PROGRAM MAIN
VAR
	AIN1 AT %I*: REAL;
	OUT AT %Q*: REAL;
	Start: BOOL;
	Stop: BOOL;
	Enable AT %Q*: BOOL;
	Home: REAL;
	Measure: REAL;
	DispSet: REAL;
		
END_VAR
VAR // added by the converter: edge detectors and wires of the graphical bodies
    _w1 : BOOL;
END_VAR

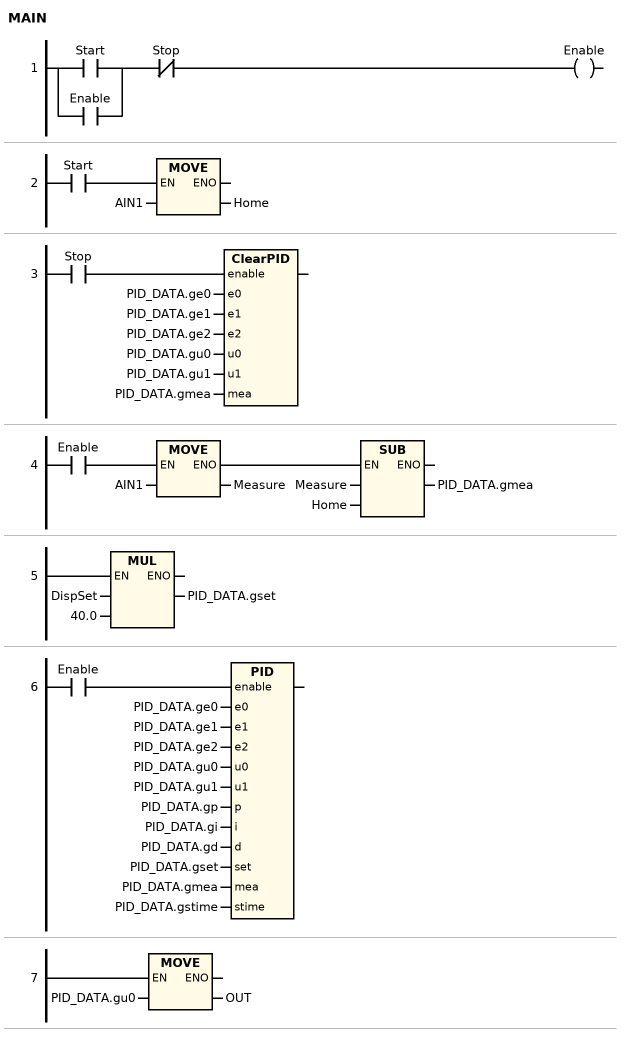
// NETWORK 1
Enable := (Start OR Enable) AND NOT Stop;

// NETWORK 2
IF Start THEN Home := AIN1; END_IF

// NETWORK 3
ClearPID(enable := Stop, e0 := PID_DATA.ge0, e1 := PID_DATA.ge1, e2 := PID_DATA.ge2, u0 := PID_DATA.gu0, u1 := PID_DATA.gu1, mea := PID_DATA.gmea);

// NETWORK 4
_w1 := Enable;
IF _w1 THEN Measure := AIN1; END_IF
IF _w1 THEN PID_DATA.gmea := Measure - Home; END_IF

// NETWORK 5
PID_DATA.gset := DispSet * 40.0;

// NETWORK 6
PID(enable := Enable, e0 := PID_DATA.ge0, e1 := PID_DATA.ge1, e2 := PID_DATA.ge2, u0 := PID_DATA.gu0, u1 := PID_DATA.gu1, p := PID_DATA.gp, i := PID_DATA.gi, d := PID_DATA.gd, set := PID_DATA.gset, mea := PID_DATA.gmea, stime := PID_DATA.gstime);

// NETWORK 7
OUT := PID_DATA.gu0;

END_PROGRAM

(* stored: Version 1.1.0.1, ProductVersion 3.1.4024.3
   POU MAIN: Id {1a862261-1045-4050-a8ea-b8696fae14b3}, SpecialFunc None *)
